PROGRAM MAIN
VAR
	
i:			INT;

END_VAR

i := i + 1;

END_PROGRAM

(* stored: Version 1.1.0.1, ProductVersion 3.1.4024.12
   POU MAIN: Id {8ccf5bf9-d764-4c6c-95fa-72dfecf03e2e}, SpecialFunc None *)
